FUNCTION_BLOCK FBD_blinker
VAR_INPUT
	execute:BOOL;
	period: TIME := T#1S;
	duty: REAL := 0.5;
END_VAR
VAR_OUTPUT
	output:BOOL;
END_VAR
VAR
	delay: TON;
END_VAR

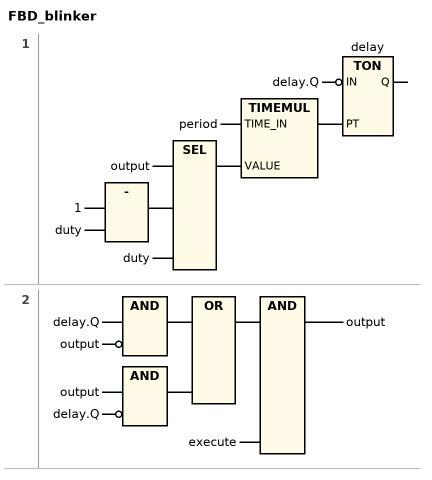
// NETWORK 1
delay(IN := NOT delay.Q, PT := TIMEMUL(TIME_IN := period, VALUE := SEL(output, 1 - duty, duty))); // TON

// NETWORK 2
output := (delay.Q AND NOT output OR output AND NOT delay.Q) AND execute;

END_FUNCTION_BLOCK

(* stored: Version 1.1.0.1, ProductVersion 3.1.4024.12
   POU FBD_blinker: Id {f2953938-7ad3-4996-bf01-3982f3a63f38}, SpecialFunc None *)
